SUBAPPLICATION Uebung_201_Interlock (* Interlock advanced exercise (AX) *)
  (* Standard: 61499-2; Description: Copyright (c) 2026 Meisterschulen am Ostbahnhof *)
  (* Version 1.0, 2026-05-07, Gemini CLI, Meisterschulen am Ostbahnhof, Interlock exercise *)
  PACKAGE Uebungen;
  IMPORT logiBUS::io::DI::logiBUS_DI::Input_I1;
  IMPORT logiBUS::io::DI::logiBUS_DI::Input_I2;
  IMPORT logiBUS::io::DI::logiBUS_DI::Input_I3;
  IMPORT logiBUS::io::DI::logiBUS_DI::Input_I4;
  IMPORT logiBUS::io::DQ::logiBUS_DO::Output_Q1;
  IMPORT logiBUS::io::DQ::logiBUS_DO::Output_Q2;
  IMPORT logiBUS::io::DQ::logiBUS_DO::Output_Q3;
  IMPORT logiBUS::io::DQ::logiBUS_DO::Output_Q4;
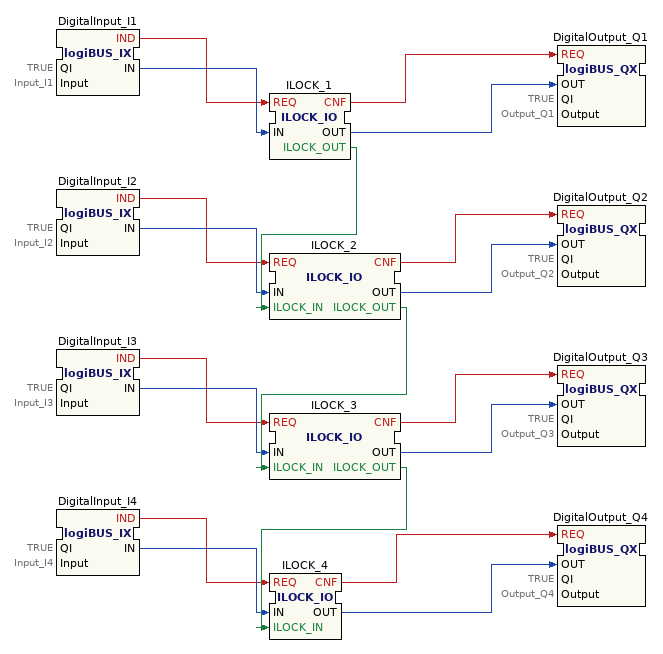
  FBS
    DigitalInput_I1 : logiBUS::io::DI::logiBUS_IX(QI := TRUE, Input := Input_I1);
    DigitalOutput_Q4 : logiBUS::io::DQ::logiBUS_QX(QI := TRUE, Output := Output_Q4);
    ILOCK_1 : logiBUS::signalprocessing::interlock::ILOCK_IO;
    DigitalInput_I2 : logiBUS::io::DI::logiBUS_IX(QI := TRUE, Input := Input_I2);
    DigitalOutput_Q1 : logiBUS::io::DQ::logiBUS_QX(QI := TRUE, Output := Output_Q1);
    ILOCK_2 : logiBUS::signalprocessing::interlock::ILOCK_IO;
    DigitalOutput_Q3 : logiBUS::io::DQ::logiBUS_QX(QI := TRUE, Output := Output_Q3);
    DigitalOutput_Q2 : logiBUS::io::DQ::logiBUS_QX(QI := TRUE, Output := Output_Q2);
    ILOCK_3 : logiBUS::signalprocessing::interlock::ILOCK_IO;
    ILOCK_4 : logiBUS::signalprocessing::interlock::ILOCK_IO;
    DigitalInput_I3 : logiBUS::io::DI::logiBUS_IX(QI := TRUE, Input := Input_I3);
    DigitalInput_I4 : logiBUS::io::DI::logiBUS_IX(QI := TRUE, Input := Input_I4);
  END_FBS
  EVENT_CONNECTIONS
    DigitalInput_I4.IND TO ILOCK_4.REQ;
    DigitalInput_I3.IND TO ILOCK_3.REQ;
    DigitalInput_I2.IND TO ILOCK_2.REQ;
    DigitalInput_I1.IND TO ILOCK_1.REQ;
    ILOCK_1.CNF TO DigitalOutput_Q1.REQ;
    ILOCK_2.CNF TO DigitalOutput_Q2.REQ;
    ILOCK_3.CNF TO DigitalOutput_Q3.REQ;
    ILOCK_4.CNF TO DigitalOutput_Q4.REQ;
  END_CONNECTIONS
  DATA_CONNECTIONS
    DigitalInput_I4.IN TO ILOCK_4.IN;
    DigitalInput_I3.IN TO ILOCK_3.IN;
    DigitalInput_I2.IN TO ILOCK_2.IN;
    DigitalInput_I1.IN TO ILOCK_1.IN;
    ILOCK_4.OUT TO DigitalOutput_Q4.OUT;
    ILOCK_3.OUT TO DigitalOutput_Q3.OUT;
    ILOCK_2.OUT TO DigitalOutput_Q2.OUT;
    ILOCK_1.OUT TO DigitalOutput_Q1.OUT;
  END_CONNECTIONS
  ADAPTER_CONNECTIONS
    ILOCK_1.ILOCK_OUT TO ILOCK_2.ILOCK_IN;
    ILOCK_2.ILOCK_OUT TO ILOCK_3.ILOCK_IN;
    ILOCK_3.ILOCK_OUT TO ILOCK_4.ILOCK_IN;
  END_CONNECTIONS
END_SUBAPPLICATION
